ABB RobotStudio station: Autoclasiffier_Vacuostato2.rspag

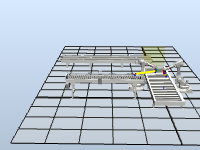
--- station ---
Station Station (saved by RobotStudio 6.6.7701.1025)
Controller Sistema12, task T_ROB1: task frame (RAPID world) sits at (920, -1100, 0) mm, rotated rx 0 ry 0 rz 180 deg in the station
Controller Sistema10, task T_ROB1: task frame (RAPID world) sits at (-920, -900, 0) mm in the station
Controller Sistema10
  mechanical unit ROB_1: JUAN, 6 joints, base frame (0, 0, 0) mm
Controller Sistema12
  mechanical unit ROB_1: ROBERTO, 6 joints, base frame (0, 0, 0) mm
Layout (positions relative to the parent item):
  - JUAN [mechanism, from Robots\IRB1600_6_145_G_02.rslib] at (-920, -900, 0) mm; joint values [-0.0666, 0.1032, 0.3482, 0, 1.1194, 3.075] (rad or m)
  - ROBERTO [mechanism, from Robots\IRB1600_6_145_G_02.rslib] at (920, -1100, 0) mm, rotated rx 0 ry 0 rz 180 deg; joint values [0.0107, 0.0331, 0.3289, -0.0129, 1.3675, 1.3261] (rad or m)
  - 600_guide [part, from Equipment\Conveyor Guide 600.rslib] at (3800, 50, 0) mm, rotated rx 0 ry 0 rz 180 deg
  - 4800_3str_h2 [part, from Equipment\Conveyor 4800 3str h2.rslib] at (0, -5364.61, 0) mm
  - 950_4800_h2 [part, from Equipment\Conveyor 950 4800 h2.rslib] at (475, -3400, 0) mm, rotated rx 0 ry 0 rz 90 deg
  - PIEZASS [part] at (920, -500, 775) mm
  - Ventosas [smart component]
      signals: DI dedo_Juan, DO Aspira, DI dedo_Roberto, DO Aspira_R
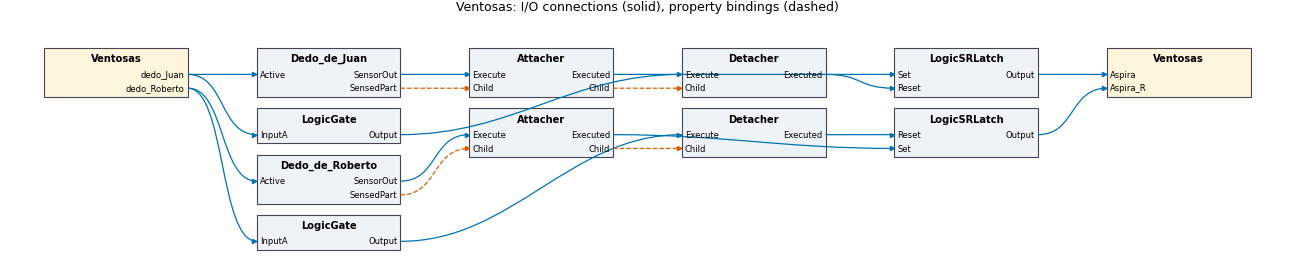
      connections:
        Dedo_de_Juan.SensorOut -> Attacher.Execute
        LogicGate.Output -> Detacher.Execute
        Ventosas.dedo_Juan -> Dedo_de_Juan.Active
        Ventosas.dedo_Juan -> LogicGate.InputA
        Attacher.Executed -> LogicSRLatch.Set
        LogicSRLatch.Output -> Ventosas.Aspira
        Detacher.Executed -> LogicSRLatch.Reset
        Ventosas.dedo_Roberto -> Dedo_de_Roberto.Active
        Dedo_de_Roberto.SensorOut -> Attacher.Execute
        LogicGate.Output -> Detacher.Execute
        Ventosas.dedo_Roberto -> LogicGate.InputA
        Detacher.Executed -> LogicSRLatch.Reset
        Attacher.Executed -> LogicSRLatch.Set
        LogicSRLatch.Output -> Ventosas.Aspira_R
        Dedo_de_Juan.SensedPart => Attacher.Child
        Attacher.Child => Detacher.Child
        Dedo_de_Roberto.SensedPart => Attacher.Child
        Attacher.Child => Detacher.Child
    - Dedo_de_Roberto [smart component, from Components\LineSensor.rslib] at (196.01, -1106.94, 909.42) mm, rotated rx -171 ry -1.53 rz -75.28 deg
        properties: Start=[0 0 0.08]; End=[0 0 0.11]; Radius=0.002; SensedPart=rueda_atras_azul; SensedPoint=[1.10435998535156 -0.361830017089844 0.9]
      - _sensorPart_ [part]
    - Attacher [smart component, from Components\Attacher.rslib]
        properties: Parent=(none); Flange=0; Child=Pieza_7; Mount=false; Offset=[0 0 0]; Orientation=[0 0 0]
    - LogicGate [smart component, from Components\LogicGate.rslib] at (-1050.67, 0, 0) mm
        properties: Operator=NOT; Delay=0
    - Dedo_de_Juan [smart component, from Components\LineSensor.rslib] at (-159.7, -950.69, 856.04) mm, rotated rx -180 ry 0 rz 0 deg
        properties: Start=[0 0 0.08]; End=[0 0 0.11]; Radius=0.002; SensedPart=Pieza_7; SensedPoint=[-0.209697967529297 -0.95068701171875 0.706042236328125]
      - _sensorPart_ [part]
    - Detacher [smart component, from Components\Detacher.rslib]
        properties: Child=Pieza_7; KeepPosition=true
    - LogicSRLatch [smart component, from Components\LogicSRLatch.rslib]
    - Attacher [smart component, from Components\Attacher.rslib]
        properties: Parent=(none); Flange=0; Child=rueda_atras_azul; Mount=false; Offset=[0 0 0]; Orientation=[0 0 0]
    - Detacher [smart component, from Components\Detacher.rslib]
        properties: Child=rueda_atras_azul; KeepPosition=true
    - LogicSRLatch [smart component, from Components\LogicSRLatch.rslib]
    - LogicGate [smart component, from Components\LogicGate.rslib]
        properties: Operator=AND; Delay=0
  - Pieza_6 [part] at (370, -1250, 415) mm, rotated rx 0 ry -90 rz 0 deg
  - T_Chasis [part] at (0, 0, 100) mm
  - Cinta_Chasis [smart component] at (0, 0, 0) mm
      signals: DI Montaje_acabado, DO Sensor, DI on
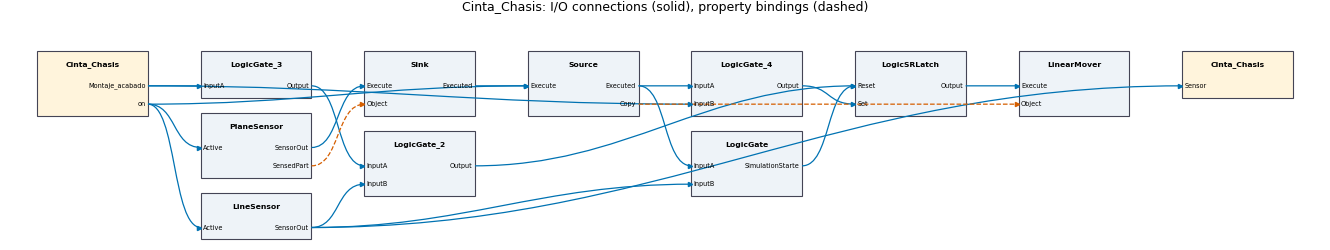
      connections:
        PlaneSensor.SensorOut -> Sink.Execute
        LogicSRLatch.Output -> LinearMover.Execute
        Source.Executed -> LogicGate.InputA
        LineSensor.SensorOut -> LogicGate.InputB
        Cinta_Chasis.Montaje_acabado -> LogicGate_3.InputA
        LogicGate_3.Output -> LogicGate_2.InputA
        LineSensor.SensorOut -> LogicGate_2.InputB
        LogicGate_2.Output -> LogicSRLatch.Reset
        Source.Executed -> LogicGate_4.InputA
        Cinta_Chasis.Montaje_acabado -> LogicGate_4.InputB
        LogicGate_4.Output -> LogicSRLatch.Set
        LineSensor.SensorOut -> Cinta_Chasis.Sensor
        Sink.Executed -> Source.Execute
        Cinta_Chasis.on -> Source.Execute
        SimulationEvents.SimulationStarted -> LogicSRLatch.Reset
        Cinta_Chasis.on -> PlaneSensor.Active
        Cinta_Chasis.on -> LineSensor.Active
        PlaneSensor.SensedPart => Sink.Object
        Source.Copy => LinearMover.Object
    - Source [smart component, from Components\Source.rslib]
        properties: Source=T_Chasis; Copy=(none); Parent=(none); Position=[0 2.5 0]; Orientation=[0 0 0]; Transient=false; PhysicsBehavior=0
    - PlaneSensor [smart component, from Components\PlaneSensor.rslib]
        properties: Origin=[-0.52 -3.6 0.35]; Axis1=[0 0 1]; Axis2=[1.05 0 0]; SensedPart=(none)
      - _sensorPart_ [part]
    - Sink [smart component, from Components\Sink.rslib]
        properties: Object=(none)
    - LinearMover [smart component, from Components\LinearMover.rslib]
        properties: Object=(none); Direction=[0 -0.001 0]; Speed=0.5; Reference=Global; ReferenceObject=(none)
    - LineSensor [smart component, from Components\LineSensor.rslib]
        properties: Start=[0.040738 -1.264377 0.404542]; End=[0.040738 -1.264377 0.42054]; Radius=0.001; SensedPart=(none); SensedPoint=[0 0 0]
      - _sensorPart_ [part]
    - LogicSRLatch [smart component, from Components\LogicSRLatch.rslib]
    - LogicGate_2 [smart component, from Components\LogicGate.rslib]
        properties: Operator=AND; Delay=0
    - LogicGate_3 [smart component, from Components\LogicGate.rslib]
        properties: Operator=NOT; Delay=0
    - LogicGate_4 [smart component, from Components\LogicGate.rslib]
        properties: Operator=OR; Delay=0
  - Mano_de_Juan [mechanism] at (-159.7, -950.69, 856.04) mm, rotated rx -180 ry 0 rz 0 deg
      TCP Mano_de_Juan at (0, 0, 100) mm
      links: Pieza_7
  - rueda_atras_azul [part] at (1106.02, -365.17, 900) mm, rotated rx 180 ry 0 rz 0 deg
  - rueda_atras_azul_2 [part] at (1107.91, -123.11, 900) mm, rotated rx 180 ry 0 rz 0 deg
  - rueda_delante_azul [part] at (1451.59, -315.99, 875) mm, rotated rx 90 ry 0 rz 0 deg
  - arandela [part] at (1451.94, -129.36, 875) mm, rotated rx 90 ry 0 rz 0 deg
  - Mano_de_Roberto [mechanism] at (196.01, -1106.94, 909.42) mm, rotated rx -171 ry -1.53 rz -75.28 deg
      TCP Mano_de_Roberto at (0, 0, 100) mm
      links: Pieza_7
  - Pieza_7 [part]
  - rueda_atras_blanca [part] at (1107.91, -123.11, 900) mm, rotated rx 180 ry 0 rz 0 deg
  - rueda_atras_blanca_2 [part] at (1106.01, -365.17, 900) mm, rotated rx 180 ry 0 rz 0 deg
  - rueda_delante_blanca [part] at (1451.59, -315.99, 875) mm, rotated rx 90 ry 0 rz 0 deg
  - rueda_atras_roja [part] at (1107.91, -123.11, 900) mm, rotated rx 180 ry 0 rz 0 deg
  - rueda_atras_roja_2 [part] at (1106.02, -365.17, 900) mm, rotated rx 180 ry 0 rz 0 deg
  - rueda_delante_roja [part] at (1451.59, -315.99, 875) mm, rotated rx 90 ry 0 rz 0 deg
  - Componente inteligente_1 [smart component]
      signals: DI on, DI fin, DO coger, DO azul, DO rojo, DO blanco
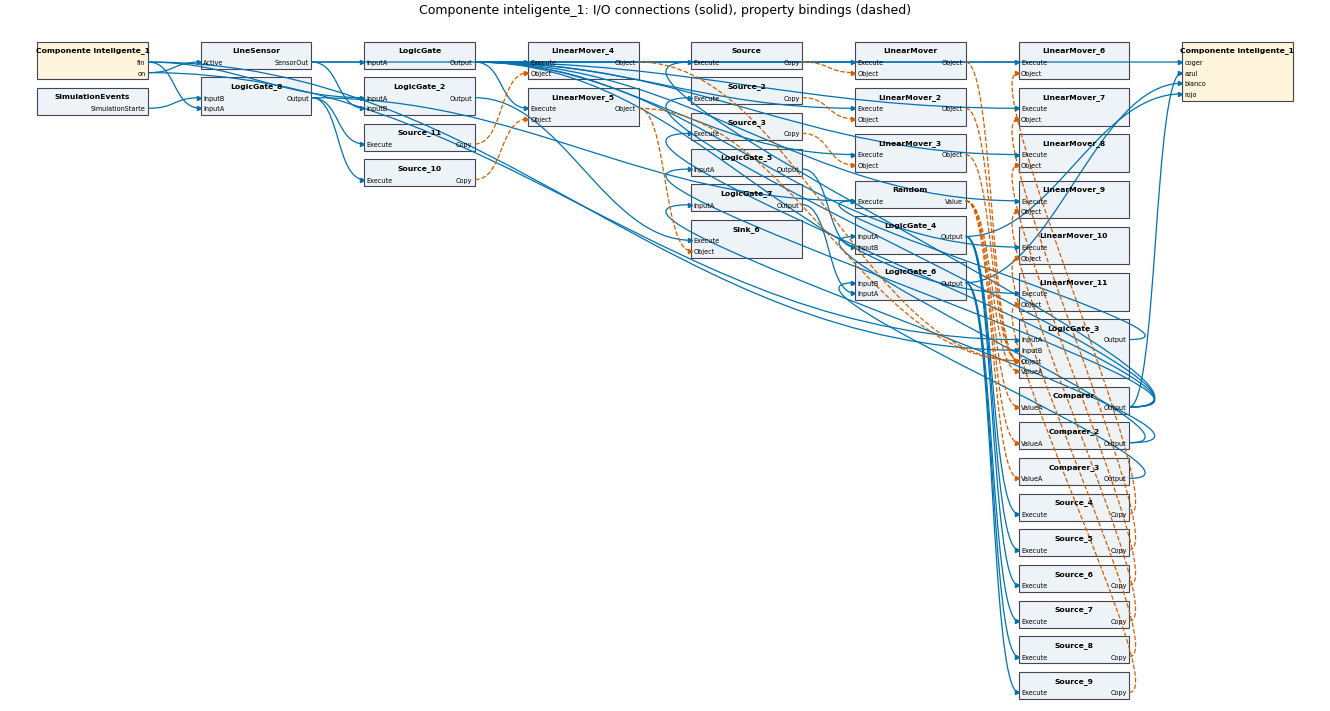
      connections:
        LineSensor.SensorOut -> LogicGate.InputA
        LogicGate.Output -> LinearMover.Execute
        LogicGate.Output -> LinearMover_2.Execute
        LogicGate.Output -> LinearMover_3.Execute
        LogicGate.Output -> LinearMover_4.Execute
        LogicGate.Output -> LinearMover_5.Execute
        Componente inteligente_1.fin -> LogicGate_2.InputA
        LineSensor.SensorOut -> LogicGate_2.InputB
        LogicGate_2.Output -> Sink_6.Execute
        Comparer.Output -> Source.Execute
        Comparer.Output -> Source_2.Execute
        Comparer.Output -> Source_3.Execute
        LogicGate.Output -> LinearMover_6.Execute
        LogicGate.Output -> LinearMover_7.Execute
        LogicGate.Output -> LinearMover_8.Execute
        LogicGate.Output -> LinearMover_9.Execute
        LogicGate.Output -> LinearMover_10.Execute
        LogicGate.Output -> LinearMover_11.Execute
        LineSensor.SensorOut -> Componente inteligente_1.coger
        Comparer.Output -> Componente inteligente_1.azul
        Componente inteligente_1.on -> LogicGate_3.InputA
        Componente inteligente_1.fin -> LogicGate_3.InputB
        LogicGate_3.Output -> Random.Execute
        Comparer_2.Output -> LogicGate_4.InputA
        LogicGate_4.Output -> Source_4.Execute
        LogicGate_4.Output -> Source_5.Execute
        LogicGate_4.Output -> Source_6.Execute
        Comparer.Output -> LogicGate_5.InputA
        LogicGate_5.Output -> LogicGate_4.InputB
        Comparer_3.Output -> LogicGate_6.InputB
        LogicGate_6.Output -> Source_7.Execute
        LogicGate_6.Output -> Source_8.Execute
        LogicGate_6.Output -> Source_9.Execute
        LogicGate_7.Output -> LogicGate_6.InputA
        LogicGate_6.Output -> Componente inteligente_1.blanco
        LogicGate_4.Output -> Componente inteligente_1.rojo
        Comparer_2.Output -> LogicGate_7.InputA
        SimulationEvents.SimulationStarted -> LogicGate_8.InputB
        Componente inteligente_1.fin -> LogicGate_8.InputA
        LogicGate_8.Output -> Source_11.Execute
        LogicGate_8.Output -> Source_10.Execute
        Componente inteligente_1.on -> LineSensor.Active
        LogicGate_8.Output -> Random.Execute
        Source.Copy => LinearMover.Object
        Source_2.Copy => LinearMover_2.Object
        Source_3.Copy => LinearMover_3.Object
        Source_11.Copy => LinearMover_4.Object
        Source_10.Copy => LinearMover_5.Object
        LinearMover.Object => Sink.Object
        LinearMover_2.Object => Sink_2.Object
        LinearMover_3.Object => Sink_3.Object
        LinearMover_4.Object => Sink_4.Object
        LinearMover_5.Object => Sink_5.Object
        LinearMover_5.Object => Sink_6.Object
        Random.Value => Comparer.ValueA
        Random.Value => Comparer_2.ValueA
        Random.Value => Comparer_3.ValueA
        Source_4.Copy => LinearMover_6.Object
        Source_5.Copy => LinearMover_7.Object
        Source_6.Copy => LinearMover_8.Object
        Source_7.Copy => LinearMover_9.Object
        Source_8.Copy => LinearMover_10.Object
        Source_9.Copy => LinearMover_11.Object
        Random.Value => Comparer_4.ValueA
    - Source [smart component, from Components\Source.rslib]
        properties: Source=rueda_atras_azul; Copy=(none); Parent=(none); Position=[3.107912 -0.123105 0.9]; Orientation=[3.14159265358979 0 0]; Transient=false; PhysicsBehavior=0
    - Source_2 [smart component, from Components\Source.rslib]
        properties: Source=rueda_atras_azul_2; Copy=(none); Parent=(none); Position=[3.106016 -0.365172 0.9]; Orientation=[3.14159265358979 0 0]; Transient=false; PhysicsBehavior=0
    - Source_3 [smart component, from Components\Source.rslib]
        properties: Source=rueda_delante_azul; Copy=(none); Parent=(none); Position=[3.451589 -0.315989 0.875]; Orientation=[1.5707963267949 0 0]; Transient=false; PhysicsBehavior=0
    - Source_4 [smart component, from Components\Source.rslib]
        properties: Source=rueda_atras_roja; Copy=(none); Parent=(none); Position=[3.107912 -0.123105 0.9]; Orientation=[3.14159265358979 0 0]; Transient=false; PhysicsBehavior=0
    - Source_5 [smart component, from Components\Source.rslib]
        properties: Source=rueda_atras_roja_2; Copy=(none); Parent=(none); Position=[3.106016 -0.365172 0.9]; Orientation=[3.14159265358979 0 0]; Transient=false; PhysicsBehavior=0
    - Source_6 [smart component, from Components\Source.rslib]
        properties: Source=rueda_delante_roja; Copy=(none); Parent=(none); Position=[3.451589 -0.315989 0.875]; Orientation=[1.5707963267949 0 0]; Transient=false; PhysicsBehavior=0
    - Source_7 [smart component, from Components\Source.rslib]
        properties: Source=rueda_atras_blanca; Copy=(none); Parent=(none); Position=[3.107912 -0.123105 0.9]; Orientation=[3.14159265358979 0 0]; Transient=false; PhysicsBehavior=0
    - Source_8 [smart component, from Components\Source.rslib]
        properties: Source=rueda_atras_blanca_2; Copy=(none); Parent=(none); Position=[3.106016 -0.365172 0.9]; Orientation=[3.14159265358979 0 0]; Transient=false; PhysicsBehavior=0
    - Source_9 [smart component, from Components\Source.rslib]
        properties: Source=rueda_delante_blanca; Copy=(none); Parent=(none); Position=[3.451589 -0.315989 0.875]; Orientation=[1.5707963267949 0 0]; Transient=false; PhysicsBehavior=0
    - Source_10 [smart component, from Components\Source.rslib]
        properties: Source=PIEZASS; Copy=(none); Parent=(none); Position=[2.92 -0.5 0.775]; Orientation=[0 0 0]; Transient=false; PhysicsBehavior=0
    - Source_11 [smart component, from Components\Source.rslib]
        properties: Source=arandela; Copy=(none); Parent=(none); Position=[3.451939 -0.129363 0.875]; Orientation=[1.5707963267949 0 0]; Transient=false; PhysicsBehavior=0
    - LineSensor [smart component, from Components\LineSensor.rslib]
        properties: Start=[0.913982 -0.348132 0.772985]; End=[0.913982 -0.348132 0.792985]; Radius=0.002; SensedPart=(none); SensedPoint=[0.913981994628906 -0.348131988525391 0.775]
      - _sensorPart_ [part]
    - LinearMover [smart component, from Components\LinearMover.rslib]
        properties: Object=(none); Direction=[-1 0 0]; Speed=0.1; Reference=Global; ReferenceObject=(none)
    - LinearMover_2 [smart component, from Components\LinearMover.rslib]
        properties: Object=(none); Direction=[-1 0 0]; Speed=0.1; Reference=Global; ReferenceObject=(none)
    - LinearMover_3 [smart component, from Components\LinearMover.rslib]
        properties: Object=(none); Direction=[-1 0 0]; Speed=0.1; Reference=Global; ReferenceObject=(none)
    - LinearMover_4 [smart component, from Components\LinearMover.rslib]
        properties: Object=(none); Direction=[-1 0 0]; Speed=0.1; Reference=Global; ReferenceObject=(none)
    - LinearMover_5 [smart component, from Components\LinearMover.rslib]
        properties: Object=(none); Direction=[-1 0 0]; Speed=0.1; Reference=Global; ReferenceObject=(none)
    - LogicGate [smart component, from Components\LogicGate.rslib]
        properties: Operator=NOT; Delay=0
    - LogicGate_2 [smart component, from Components\LogicGate.rslib]
        properties: Operator=AND; Delay=0
    - Sink_6 [smart component, from Components\Sink.rslib]
        properties: Object=(none)
    - Random [smart component, from Components\Random.rslib]
        properties: Value=2.87996190827338; Min=0; Max=3
    - Comparer [smart component, from Components\Comparer.rslib]
        properties: ValueA=2.87996190827338; Operator=<=; ValueB=1
    - Comparer_2 [smart component, from Components\Comparer.rslib]
        properties: ValueA=2.87996190827338; Operator=<=; ValueB=2
    - Comparer_3 [smart component, from Components\Comparer.rslib]
        properties: ValueA=2.87996190827338; Operator=<=; ValueB=3
    - LinearMover_6 [smart component, from Components\LinearMover.rslib]
        properties: Object=(none); Direction=[-1 0 0]; Speed=0.1; Reference=Global; ReferenceObject=(none)
    - LinearMover_7 [smart component, from Components\LinearMover.rslib]
        properties: Object=(none); Direction=[-1 0 0]; Speed=0.1; Reference=Global; ReferenceObject=(none)
    - LinearMover_8 [smart component, from Components\LinearMover.rslib]
        properties: Object=(none); Direction=[-1 0 0]; Speed=0.1; Reference=Global; ReferenceObject=(none)
    - LinearMover_9 [smart component, from Components\LinearMover.rslib]
        properties: Object=(none); Direction=[-1 0 0]; Speed=0.1; Reference=Global; ReferenceObject=(none)
    - LinearMover_10 [smart component, from Components\LinearMover.rslib]
        properties: Object=(none); Direction=[-1 0 0]; Speed=0.1; Reference=Global; ReferenceObject=(none)
    - LinearMover_11 [smart component, from Components\LinearMover.rslib]
        properties: Object=(none); Direction=[-1 0 0]; Speed=0.1; Reference=Global; ReferenceObject=(none)
    - Converter [smart component, from Components\Converter.rslib]
        properties: AnalogProperty=0; DigitalProperty=0; BooleanProperty=false; GroupProperty=0
    - LogicGate_4 [smart component, from Components\LogicGate.rslib]
        properties: Operator=AND; Delay=0
    - LogicGate_5 [smart component, from Components\LogicGate.rslib]
        properties: Operator=NOT; Delay=0
    - LogicGate_6 [smart component, from Components\LogicGate.rslib]
        properties: Operator=AND; Delay=0
    - LogicGate_7 [smart component, from Components\LogicGate.rslib]
        properties: Operator=NOT; Delay=0
    - SimulationEvents [smart component, from Components\SimulationEvents.rslib]
    - LogicGate_8 [smart component, from Components\LogicGate.rslib]
        properties: Operator=OR; Delay=0
  - Pieza_8 [part]
Attachment: Mano_de_Juan is attached to JUAN / Link6
Attachment: Dedo_de_Juan is attached to Mano_de_Juan / Pieza_7
Attachment: Mano_de_Roberto is attached to ROBERTO / Link6
Attachment: Dedo_de_Roberto is attached to Mano_de_Roberto / Pieza_7
Attachment: Cinta_Chasis is attached to Mano_de_Juan / Pieza_7
Station logic (signal -> signal, property => property):
  Ventosas.Aspira -> Sistema10.PiezaCogida_Juan
  Sistema10.ActivaMano_Juan -> Ventosas.dedo_Juan
  Sistema10.Cinta_on -> Cinta_Chasis.on
  Sistema10.Montaje_fin -> Cinta_Chasis.Montaje_acabado
  Sistema12.ActivaMano_Roberto -> Ventosas.dedo_Roberto
  Ventosas.Aspira_R -> Sistema12.PiezaCogida_Roberto
  Sistema12.PiezaColocada -> Sistema10.PiezaColocada
  Cinta_Chasis.Sensor -> Sistema12.Sensor_cinta1
  Sistema12.cinta2_on -> Componente inteligente_1.on
  Sistema12.fin_piezas -> Componente inteligente_1.fin
  Componente inteligente_1.coger -> Sistema12.Piezas_listas
  Cinta_Chasis.Sensor -> Sistema10.Sensor_cinta10
Targets, tools, work objects and paths stored in the station and not in the controller backup, written as RAPID:
! task T_ROB1
MODULE Module1
  CONST robtarget Target_10:=[[710.302,-50.687,666.042],[0,1,0,0],[-1,0,1,0],[9E+09,9E+09,9E+09,9E+09,9E+09,9E+09]];
  CONST robtarget Target_20:=[[760.301980587,-50.686989693,756.042035513],[-0.000000033,1,-0.000000027,0.000000018],[-1,-1,1,0],[9E+09,9E+09,9E+09,9E+09,9E+09,9E+09]];
ENDMODULE

! task T_ROB1
MODULE Module1
  CONST robtarget Target_10:=[[-184.36,-738.17,893],[0,1,0,0],[-2,0,0,0],[9E+09,9E+09,9E+09,9E+09,9E+09,9E+09]];
  CONST robtarget Target_20:=[[708.18882541,5.505341968,810.681077106],[0.058416761,-0.607911824,-0.790008473,0.054012115],[0,-1,0,0],[9E+09,9E+09,9E+09,9E+09,9E+09,9E+09]];
ENDMODULE


--- Backups/Sistema10/RAPID/TASK1/PROGMOD/CalibData.mod ---
MODULE CalibData
	PERS tooldata Ventosa1:=[TRUE,[[0.000009563,-0.000007568,35],[1,0,0,0]],[1,[0,0,1],[1,0,0,0],0,0,0]];
	PERS tooldata Mano_de_Juan:=[TRUE,[[0,0,100],[1,0,0,0]],[1,[0,0,1],[1,0,0,0],0,0,0]];
ENDMODULE

--- Backups/Sistema10/RAPID/TASK1/PROGMOD/Module1.mod ---
MODULE Module1
		VAR bool i:=FALSE;
        CONST robtarget RuedaTrasera1_Pos2:=[[710,60,695],[0.707106781,0.707106781,0,0],[-2,-1,0,7],[9E+09,9E+09,9E+09,9E+09,9E+09,9E+09]];
	    VAR robtarget RT1_P2;

    PROC Atornilla()
        RT1_P2:=RelTool(RuedaTrasera1_Pos2,0,0,-25);

            SetDO ActivaMano_Juan,0;
            SetDO ActivaMano_Juan,1;
            WaitRob \ZeroSpeed;
        SetDO ActivaMano_Juan,0;
        MoveL RuedaTrasera1_Pos2,v100,z100,Mano_de_Juan\WObj:=wobj0;
            WaitRob \ZeroSpeed;
            WaitRob \ZeroSpeed;
            SetDO ActivaMano_Juan,1;
        MoveL RuedaTrasera1_Pos2,v100,z100,Mano_de_Juan\WObj:=wobj0;
            WaitRob \ZeroSpeed;
            SetDO ActivaMano_Juan,0;
	ENDPROC

PROC INICIO()

        IF i=FALSE THEN
        SetDO Cinta_on,0;
        WaitTime 1;
        SetDO Cinta_on,1;
        i:=TRUE;
        ENDIF

ENDPROC

    PROC main()

        SetDO Montaje_fin,1;
        SetDO Montaje_fin,0;
        INICIO;
        WaitDI PiezaColocada,0;
        WaitDI PiezaColocada,1;
        Atornilla;
        WaitTime 1;
        SetDO  Montaje_fin,1;
        WaitDI Sensor_cinta10,0;
        SetDO  Montaje_fin,0;



    ENDPROC

ENDMODULE

--- Backups/Sistema10/RAPID/TASK1/SYSMOD/LINKEDM.sys ---
%%%
  VERSION:1
  LANGUAGE:ENGLISH
%%%

MODULE LINKEDM (SYSMODULE)

! FOLLOWER
!     Name of electronically linked follower axis used by operator at teach pendent.
      PERS string l_f_axis_name{5}       :=  ["",  "", "", "", ""];

!     Name of the mechanical unit for follower axis.
      PERS string l_f_mecunt_n{5}  :=  ["", "", "", "", ""];

!     Linked follower axis number in the mechanical unit (first axis in mech. unit is number 1).
      PERS num l_f_axis_no{5}      :=  [0,          0,   0,  0,  0];

! MASTER
!     Name of the mechanical unit for linked master axis.
      PERS string l_m_mecunt_n{5} :=  ["", "", "", "", ""];

!     Linked master axis number in the mechanical unit (first axis in mech. unit is number 1).
!     See axis number table in documentation for different master mechanical units.
      PERS num l_m_axis_no{5}     :=  [0,  0,  0,  0,  0];

! POSITION OFFSET
!     The increase of the allowed offset position between the master and follower
!     positions, used when starting AUTO mode. As soon as the offset is decreased
!     the old configurated parameter is used.
!     Example: 3 => the configurated value of allowed offset is increased 3 times.
      PERS num offset_ratio{5}       :=  [10,  10,   10,  10,  10];

! SPEED RATIO
!     Speed_ratio used in AUTO and JOG modes [ very_slow   slow    normal    fast]
!     Value 1 = max allowed manual speed.
      CONST num speed_ratio {20}      := [0.01, 0.01, 0.01, 0.01, 0.01,
                                          0.05, 0.05, 0.05, 0.05, 0.05,
                                          0.20, 0.20, 0.20, 0.20, 0.20,
                                          1.00, 1.00, 1.00, 1.00, 1.00];

! STEP SIZE
!     Displacement position used in JOG mode for each activation of positive or
!     negative movement.                  [very_short    short   normal   long]
!     Unit degees or meter.
      CONST num displacement {20}     := [0.001, 0.001, 0.001, 0.001, 0.001,
                                          0.005, 0.005, 0.005, 0.005, 0.005,
                                          0.020, 0.020, 0.020, 0.020, 0.020,
                                          0.100, 0.100, 0.100, 0.100, 0.100];


!-------------------------------------------------------------
 PROC Linked_m ()
      Linked_m_exe ;
 ENDPROC
ENDMODULE

--- Backups/Sistema12/RAPID/TASK1/PROGMOD/CalibData.mod ---
MODULE CalibData
	PERS tooldata Mano_de_Roberto:=[TRUE,[[0,0,100],[1,0,0,0]],[1,[0,0,1],[1,0,0,0],0,0,0]];
ENDMODULE

--- Backups/Sistema12/RAPID/TASK1/PROGMOD/Module1.mod ---
MODULE Module1
	CONST robtarget RuedaTrasera1_Pos1:=[[-186.016,-734.828,902.5],[0,1,0,0],[-2,0,0,0],[9E+09,9E+09,9E+09,9E+09,9E+09,9E+09]];
	CONST robtarget RuedaTrasera1_Pos2:=[[1130,-260,695],[0,0,0.707106781,0.707106781],[-1,0,-1,0],[9E+09,9E+09,9E+09,9E+09,9E+09,9E+09]];
	VAR robtarget RT1_P1;
    VAR robtarget RT1_P2;
    VAR bool i:=FALSE;



    PROC TrasladoPiezas()

        RT1_P1:=RelTool(RuedaTrasera1_Pos1,0,0,-30);
        RT1_P2:=RelTool(RuedaTrasera1_Pos2,0,0,-25);

            SetDO PiezaColocada,0;
            SetDO ActivaMano_Roberto,0;

	    MoveJ RuedaTrasera1_Pos1,v100,z100,Mano_de_Roberto\WObj:=wobj0;
            WaitRob \ZeroSpeed;
            SetDO ActivaMano_Roberto,1;
        MoveL RT1_P1,v1000,z100,Mano_de_Roberto\WObj:=wobj0;
        MoveJ RT1_P2,v1000,z100,Mano_de_Roberto\WObj:=wobj0;
             WaitRob \ZeroSpeed;
             SetDO ActivaMano_Roberto,0;
             SetDO PiezaColocada,1;
        MoveJ RT1_P1,v1000,z100,Mano_de_Roberto\WObj:=wobj0;



	ENDPROC

    PROC INICIO()

        IF i=FALSE THEN
        SetDO cinta2_on,0;
        WaitTime 1;
        SetDO cinta2_on,1;
        i:=TRUE;
        ENDIF

ENDPROC

    PROC main()
        INICIO;
        WaitDI Piezas_listas,1;
        WaitTime 3;
        !WaitDI Sensor_cinta1,0;
        WaitDI Sensor_cinta1,1;
        TrasladoPiezas;



    ENDPROC
    PROC Path_10()
        MoveJ RuedaTrasera1_Pos1,v1000,z100,Mano_de_Roberto\WObj:=wobj0;
        MoveJ RuedaTrasera1_Pos2,v1000,z100,Mano_de_Roberto\WObj:=wobj0;
    ENDPROC
ENDMODULE

--- Backups/Sistema10/SYSPAR/EIO.cfg ---
EIO:CFG_1.0:6:1::
#
INDUSTRIAL_NETWORK:

      -Name "DeviceNet" -Label "DeviceNet Master/Slave Network" -Address "2"
#
DEVICENET_DEVICE:

      -Name "ModuloES" -Simulated
#
DEVICENET_INTERNAL_DEVICE:

      -Name "DN_Internal_Device" -VendorName "ABB Robotics"\
      -ProductName "DeviceNet Internal Slave Device"
#
EIO_SIGNAL:

      -Name "PiezaCogida_Juan" -SignalType "DI" -Device "ModuloES"\
      -Label "PiezaCogida_Juan" -DeviceMap "0" -Access "All"

      -Name "ActivaMano_Juan" -SignalType "DO" -Device "ModuloES"\
      -Label "ActivaMano_Juan" -DeviceMap "0" -Access "All"

      -Name "Cinta_on" -SignalType "DO" -Device "ModuloES" -Label "Cinta_on"\
      -DeviceMap "1" -Access "All"

      -Name "Sensor_cinta10" -SignalType "DI" -Device "ModuloES"\
      -Label "Sensor_cinta10" -DeviceMap "1" -Access "All"

      -Name "Montaje_fin" -SignalType "DO" -Device "ModuloES"\
      -Label "Montaje_fin" -DeviceMap "2" -Access "All"

      -Name "PiezaColocada" -SignalType "DI" -Device "ModuloES"\
      -Label "PiezaColocada" -DeviceMap "2" -Access "All"

--- Backups/Sistema12/SYSPAR/EIO.cfg ---
EIO:CFG_1.0:6:1::
#
INDUSTRIAL_NETWORK:

      -Name "DeviceNet" -Label "DeviceNet Master/Slave Network" -Address "2"\
      -Simulated
#
DEVICENET_DEVICE:

      -Name "ModuloES" -Simulated
#
DEVICENET_INTERNAL_DEVICE:

      -Name "DN_Internal_Device" -VendorName "ABB Robotics"\
      -ProductName "DeviceNet Internal Slave Device"
#
EIO_SIGNAL:

      -Name "ActivaMano_Roberto" -SignalType "DO" -Device "ModuloES"\
      -Label "ActivaMano_Roberto" -DeviceMap "0" -Access "All"

      -Name "PiezaCogida_Roberto" -SignalType "DI" -Device "ModuloES"\
      -Label "PiezaCogida_Roberto" -DeviceMap "0" -Access "All"

      -Name "Sensor_cinta1" -SignalType "DI" -Device "ModuloES"\
      -Label "Sensor_cinta1" -DeviceMap "2" -Access "All"

      -Name "PiezaColocada" -SignalType "DO" -Device "ModuloES"\
      -Label "PiezaColocada" -DeviceMap "2" -Access "All"

      -Name "cinta2_on" -SignalType "DO" -Device "ModuloES" -Label "cinta2_on"\
      -DeviceMap "3" -Access "All"

      -Name "fin_piezas" -SignalType "DO" -Device "ModuloES" -Label "fin_piezas"\
      -DeviceMap "4" -Access "All"

      -Name "Piezas_listas" -SignalType "DI" -Device "ModuloES"\
      -Label "Piezas_listas" -DeviceMap "4" -Access "All"
